// TwinCAT 3 PLC project SystemControl
// Title: Tk_SystemControl
// Company: Komatsu
// Author: TK
// ProjectVersion: 0.0.5.0
// Description: システムの管理用ライブラリ パーシステントデータ管理、PC電源管理
// ProgramVersion: 3.1.4026.26
// libraries:
//   Tc2_IoFunctions, * (Beckhoff Automation GmbH)
//   Tc2_Standard, * (Beckhoff Automation GmbH)
//   Tc2_SUPS, * (Beckhoff Automation GmbH)
//   Tc2_System, * (Beckhoff Automation GmbH)
//   Tc2_Utilities, * (Beckhoff Automation GmbH)
//   Tc3_EventLogger, * (Beckhoff Automation GmbH)
// project tree:
//   PcPower/1s_UPS/ FB_1s_UPS_BAPI.TcPOU, FB_1s_UPS_Base.TcPOU, FB_1s_UPS_CX81xx.TcPOU, I_1s_UPS.TcIO
//   PcPower/ FB_PcShutdownController.TcPOU
//   PcPower/UPS/ FB_UPS_Base.TcPOU, FB_UPS_CU81x0_0xx0.TcPOU, I_UPS.TcIO
//   PcPower/[obsolete]/1sUPS/ FB_1sUPS_BAPI.TcPOU, FB_1sUPS_CX81xx.TcPOU, i1sUPS.TcIO
//   PcPower/[obsolete]/ FB_PcPowerManagement.TcPOU
//   PersistentData/ FB_PersistentDataManager.TcPOU (not stored)
//   PersistentData/[obsolete]/ FB_PersistentDataManagement.TcPOU (not stored)
//   Version/ Global_Version.TcGVL
// (motion and I/O tree: see PLC project wago7871664000080)
// real-time tasks:
//   TASK PlcTask: cycle T#10ms, priority 20, ADS port 350

// ---- Version/Global_Version.TcGVL
{attribute 'TcGenerated'}
{attribute 'no-analysis'}
{attribute 'linkalways'}
// This function has been automatically generated from the project information.
VAR_GLOBAL CONSTANT
	{attribute 'const_non_replaced'}
	stLibVersion_Tk_SystemControl : ST_LibVersion := (iMajor := 0, iMinor := 0, iBuild := 5, iRevision := 0, nFlags := 0, sVersion := '0.0.5.0');
END_VAR

// ---- PcPower/1s_UPS/I_1s_UPS.TcIO
INTERFACE I_1s_UPS

METHOD AcknowledgePowerFailDetect
VAR_INPUT
END_VAR
END_METHOD

PROPERTY bPowerFailDetect : BOOL
GET
END_GET
END_PROPERTY

PROPERTY bReady : BOOL
GET
END_GET
END_PROPERTY

PROPERTY e1sUpsState : E_S_UPS_State
GET
END_GET
END_PROPERTY

METHOD Execute
VAR_INPUT
END_VAR
END_METHOD

//FB_Init は常に暗黙的に使用可能で、主に初期化に使用されます。
//戻り値は評価されません。特定の結果を得るために、メソッドを明示的に宣言し、
//そのメソッドに標準の初期化コードをもったコードを追加することができます。戻り値を評価できます。
METHOD FB_Init: BOOL
VAR_INPUT
    bInitRetains: BOOL; // TRUE: 保持変数は初期化されます (ウォーム リセット、あるいはコールド リセット)
    bInCopyCode: BOOL;  // TRUE: 後でコードをコピーする (オンライン変更) ために、インスタンスをコピーします。

	PcAmsNetId					:AMSNETID;		//PC AMS Net ID
END_VAR
END_METHOD

END_INTERFACE

// ---- PcPower/UPS/I_UPS.TcIO
INTERFACE I_UPS

METHOD AcknowledgePowerFailDetect
VAR_INPUT
END_VAR
END_METHOD

PROPERTY bPowerFailDetect : BOOL
GET
END_GET
END_PROPERTY

PROPERTY bReady : BOOL
GET
END_GET
END_PROPERTY

PROPERTY bReplaceBattery : BOOL
GET
END_GET
END_PROPERTY

METHOD Execute
VAR_INPUT
END_VAR
END_METHOD

//FB_Init は常に暗黙的に使用可能で、主に初期化に使用されます。
//戻り値は評価されません。特定の結果を得るために、メソッドを明示的に宣言し、
//そのメソッドに標準の初期化コードをもったコードを追加することができます。戻り値を評価できます。
METHOD FB_Init: BOOL
VAR_INPUT
    bInitRetains: BOOL; // TRUE: 保持変数は初期化されます (ウォーム リセット、あるいはコールド リセット)
    bInCopyCode: BOOL;  // TRUE: 後でコードをコピーする (オンライン変更) ために、インスタンスをコピーします。

	PcAmsNetId					:AMSNETID;		//PC AMS Net ID
END_VAR
END_METHOD

PROPERTY nBatteryPercent : DWORD
GET
END_GET
END_PROPERTY

END_INTERFACE

// ---- PcPower/[obsolete]/1sUPS/i1sUPS.TcIO
INTERFACE i1sUPS

PROPERTY bPowerFailDetect : bool
GET
END_GET
END_PROPERTY

PROPERTY eUpsState : E_S_UPS_State
GET
END_GET
END_PROPERTY

METHOD UPSCall
VAR_INPUT
	(*PC AMS Net ID*)
	PcAmsNetId	: AMSNETID;
END_VAR
END_METHOD

END_INTERFACE

// ---- PcPower/1s_UPS/FB_1s_UPS_BAPI.TcPOU
FUNCTION_BLOCK FB_1s_UPS_BAPI EXTENDS FB_1s_UPS_Base
VAR CONSTANT
	nOkCapacityLevel	:BYTE	:=90;
END_VAR
VAR
	fb1sUps				:FB_S_UPS_BAPI;
END_VAR

METHOD Execute
fb1sUps(sNetID				:=F_CreateAmsNetId(_PcAmsNetId),
		iPLCPort			:=TwinCAT_SystemInfoVarList._AppInfo.AdsPort,
		tTimeout			:=DEFAULT_ADS_TIMEOUT,
		eUpsMode			:=E_S_UPS_Mode.eSUPS_WrPersistData_Shutdown,
		ePersistentMode		:=E_PersistentMode.SPDM_2PASS,
		tRecoverTime		:=T#10S,
		bPowerFailDetect	=>,
		eState				=>SUPER^._e1sUpsState,
		nCapacity			=>,
		bBusy				=>,
		bError				=>,
		nErrID				=>
		);
		
IF fb1sUps.bPowerFailDetect THEN
	SUPER^._bPowerFailDetect:=TRUE;
END_IF

SUPER^._bReady:=(fb1sUps.eState=E_S_UPS_State.eSUPS_PowerOK) AND (nOkCapacityLevel<fb1sUps.nCapacity) AND (fb1sUps.bError=FALSE);
END_METHOD

END_FUNCTION_BLOCK

// ---- PcPower/1s_UPS/FB_1s_UPS_Base.TcPOU
FUNCTION_BLOCK FB_1s_UPS_Base IMPLEMENTS I_1s_UPS
VAR
	_PcAmsNetId				:AMSNETID;			//PC AMS Net ID	
	
	_bReady					:BOOL;				//電源供給あり
	_e1sUpsState			:E_S_UPS_State;		//1s UPSのステータス
	
	{attribute 'TcPersistent'}
	_bPowerFailDetect		:BOOL;				//停電検知記憶
END_VAR

METHOD AcknowledgePowerFailDetect
_bPowerFailDetect:=FALSE;
END_METHOD

PROPERTY bPowerFailDetect : BOOL
GET
bPowerFailDetect:=_bPowerFailDetect;
END_GET
END_PROPERTY

PROPERTY bReady : BOOL
GET
bReady:=_bReady;
END_GET
END_PROPERTY

PROPERTY e1sUpsState : E_S_UPS_State
GET
e1sUpsState:=_e1sUpsState;
END_GET
END_PROPERTY

METHOD Execute
END_METHOD

//FB_Init は常に暗黙的に使用可能で、主に初期化に使用されます。
//戻り値は評価されません。特定の結果を得るために、メソッドを明示的に宣言し、
//そのメソッドに標準の初期化コードをもったコードを追加することができます。戻り値を評価できます。
METHOD FB_Init: BOOL
VAR_INPUT
    bInitRetains: BOOL; // TRUE: 保持変数は初期化されます (ウォーム リセット、あるいはコールド リセット)
    bInCopyCode: BOOL;  // TRUE: 後でコードをコピーする (オンライン変更) ために、インスタンスをコピーします。

	PcAmsNetId					:AMSNETID;		//PC AMS Net ID
END_VAR
_PcAmsNetId:=PcAmsNetId;
END_METHOD

END_FUNCTION_BLOCK

// ---- PcPower/1s_UPS/FB_1s_UPS_CX81xx.TcPOU
FUNCTION_BLOCK FB_1s_UPS_CX81xx EXTENDS FB_1s_UPS_Base
VAR
	fb1sUps		:FB_S_UPS_CX81xx;
END_VAR

METHOD Execute
fb1sUps(sNetID				:=F_CreateAmsNetId(_PcAmsNetId),
		iPLCPort			:=TwinCAT_SystemInfoVarList._AppInfo.AdsPort,
		tTimeout			:=DEFAULT_ADS_TIMEOUT,
		eUpsMode			:=E_S_UPS_Mode.eSUPS_WrPersistData_Shutdown,
		ePersistentMode		:=E_PersistentMode.SPDM_2PASS,
		tRecoverTime		:=T#10S,
		bPowerFailDetect	=>,
		eState				=>SUPER^._e1sUpsState
		);

IF fb1sUps.bPowerFailDetect THEN
	SUPER^._bPowerFailDetect:=TRUE;
END_IF

SUPER^._bReady:= fb1sUps.eState=E_S_UPS_State.eSUPS_PowerOK;
END_METHOD

END_FUNCTION_BLOCK

// ---- PcPower/FB_PcShutdownController.TcPOU
FUNCTION_BLOCK FB_PcShutdownController
VAR
//---FB_Initで受け取り---
	_pPersistentDataManager		:POINTER TO FB_PersistentDataManager;		//パーシステントデータ書き込み
	_PcAmsNetId					:AMSNETID;									//PC AMS Net ID	

//---内部使用FB---
	fbPlcStop					:PLC_Stop		:=(Stop:=FALSE);			//PLCストップ
	fbNtShutdown				:NT_Shutdown	:=(START:=FALSE);			//PCシャットダウン
	fbNtReboot					:NT_Reboot		:=(START:=FALSE);			//PCリブート

	fbRebootTon					:TON			:=(PT:=T#2S);
	fbShutdownTon				:TON			:=(PT:=T#2S);
	
//---内部変数---
	iStep						:INT			:=0;						//シャットダウン、リブート制御step
	_bError						:BOOL;
	_bReboot					:BOOL;
	_bShutdown					:BOOL;
END_VAR

PROPERTY bError : BOOL
GET
bError:=_bError;
END_GET
END_PROPERTY

METHOD Execute
//---パーシステントデータ保存FBのポインターチェック---
	IF _pPersistentDataManager=0 THEN
		_bError:=TRUE;
		iStep:=0;
		RETURN;
		
	END_IF	



//---タイマーFB呼び出し---
	fbRebootTon(IN:=_bReboot AND NOT _bShutdown AND NOT _bError );
	fbShutdownTon(IN:=_bShutdown AND NOT _bReboot AND NOT _bError );



//---制御step---
	CASE iStep OF
		0:
			IF fbRebootTon.Q OR fbShutdownTon.Q THEN
				iStep:=10;
				
			END_IF
			
		10:				
			_pPersistentDataManager^.RequestWrite();
			iStep:=20;
	
		20:
			IF _pPersistentDataManager^.bWritePersistentDataDone THEN
				iStep:=30;
			ELSIF _pPersistentDataManager^.bWritePersistentDataError THEN
				_bError:=TRUE;
				iStep:=0;
			END_IF
		
		30:
		(*	fbPlcStop(	NETID	:=F_CreateAmsNetId(_PcAmsNetId),
						PORT	:=TwinCAT_SystemInfoVarList._AppInfo.AdsPort,
						Stop	:=_bReboot OR _bShutdown,
						TMOUT	:=DEFAULT_ADS_TIMEOUT,
						BUSY	=>,
						ERR		=>,
						ERRID	=>
						);
		*)
		
			fbNtReboot(	NETID	:=F_CreateAmsNetId(_PcAmsNetId),
						DELAY	:=1,
						START	:=_bReboot,
						TMOUT	:=DEFAULT_ADS_TIMEOUT,
						BUSY	=>,
						ERR		=>,
						ERRID	=>
						);
		
			fbNtShutdown(	NETID	:=F_CreateAmsNetId(_PcAmsNetId),
							DELAY	:=1,
							START	:=_bShutdown,
							TMOUT	:=DEFAULT_ADS_TIMEOUT,
							BUSY	=>,
							ERR		=>,
							ERRID	=>
							);
	
	END_CASE
END_METHOD

//FB_Init は常に暗黙的に使用可能で、主に初期化に使用されます。
//戻り値は評価されません。特定の結果を得るために、メソッドを明示的に宣言し、
//そのメソッドに標準の初期化コードをもったコードを追加することができます。戻り値を評価できます。
METHOD FB_Init: BOOL
VAR_INPUT
    bInitRetains: BOOL; // TRUE: 保持変数は初期化されます (ウォーム リセット、あるいはコールド リセット)
    bInCopyCode: BOOL;  // TRUE: 後でコードをコピーする (オンライン変更) ために、インスタンスをコピーします。

    pPersistentDataManager		:POINTER TO FB_PersistentDataManager;
	PcAmsNetId					:AMSNETID;		//PC AMS Net ID
END_VAR
_pPersistentDataManager := pPersistentDataManager;

_PcAmsNetId:=PcAmsNetId;
END_METHOD

METHOD  RequestReboot: BOOL
VAR_INPUT
	bExecute	:bool;
END_VAR
_bReboot		:=bExecute;
RequestReboot	:=bExecute;
END_METHOD

METHOD RequestShutdown: BOOL
VAR_INPUT
	bExecute	:BOOL;
END_VAR
_bShutdown			:=bExecute;
RequestShutdown		:=bExecute;
END_METHOD

METHOD ResetError
//エラー出力をリセット
_bError:=FALSE;
END_METHOD

END_FUNCTION_BLOCK

// ---- PcPower/UPS/FB_UPS_Base.TcPOU
FUNCTION_BLOCK FB_UPS_Base IMPLEMENTS I_UPS
VAR
	_PcAmsNetId				:AMSNETID;			//PC AMS Net ID	
	
	_bReady					:BOOL;				//電源供給あり
	_bReplaceBattery		:BOOL;				//バッテリー寿命・交換警告
	
	_nBatteryPercent		:DWORD;				//バッテリー残量 (0-100%)
	
	{attribute 'TcPersistent'}
	_bPowerFailDetect		:BOOL;				//停電検知記憶
END_VAR

METHOD AcknowledgePowerFailDetect
_bPowerFailDetect:=FALSE;
END_METHOD

PROPERTY bPowerFailDetect : BOOL
GET
bPowerFailDetect:=_bPowerFailDetect;
END_GET
END_PROPERTY

PROPERTY bReady : BOOL
GET
bReady:=_bReady;
END_GET
END_PROPERTY

PROPERTY bReplaceBattery : BOOL
GET
bReplaceBattery:=_bReplaceBattery;
END_GET
END_PROPERTY

METHOD Execute
END_METHOD

(*FB_Init は常に暗黙的に使用可能で、主に初期化に使用されます。
戻り値は評価されません。特定の結果を得るために、メソッドを明示的に宣言し、
そのメソッドに標準の初期化コードをもったコードを追加することができます。戻り値を評価できます。*)
METHOD FB_Init : BOOL
VAR_INPUT
	(* TRUE: 保持変数は初期化されます (ウォーム リセット、あるいはコールド リセット)*)
	bInitRetains	: BOOL;
	(* TRUE: 後でコードをコピーする (オンライン変更) ために、インスタンスをコピーします。*)
	bInCopyCode	: BOOL;
	(*PC AMS Net ID*)
	PcAmsNetId	: AMSNETID;
END_VAR
_PcAmsNetId:=PcAmsNetId;
END_METHOD

PROPERTY nBatteryPercent : DWORD
GET
nBatteryPercent:=_nBatteryPercent;
END_GET
END_PROPERTY

END_FUNCTION_BLOCK

// ---- PcPower/UPS/FB_UPS_CU81x0_0xx0.TcPOU
FUNCTION_BLOCK FB_UPS_CU81x0_0xx0 EXTENDS FB_UPS_Base
VAR_INPUT
END_VAR
VAR_OUTPUT
END_VAR
VAR
	fbUps			:FB_GetUPSStatus;
	_stUpsStatus	:ST_UPSStatus;
END_VAR

METHOD Execute
fbUps(	sNetId		:=SUPER^._PcAmsNetId,
		nPort		:=0,
		bEnable		:=TRUE,
		bValid		=>,
		bError		=>,
		nErrId		=>,
		stStatus	=>_stUpsStatus
		);

SUPER^._bReady:= fbUps.stStatus.ePowerStatus=E_UpsPowerStatus.PowerOnLine;

SUPER^._bPowerFailDetect:= fbUps.stStatus.ePowerStatus=E_UpsPowerStatus.PowerOnBattery;

SUPER^._bReplaceBattery:=fbUps.stStatus.eBatteryStatus=E_BatteryStatus.BatteryReplace;

SUPER^._nBatteryPercent:=fbUps.stStatus.BatteryLifePercent;
END_METHOD

PROPERTY stUpsStatus : ST_UPSStatus
GET
stUpsStatus:=_stUpsStatus;
END_GET
END_PROPERTY

END_FUNCTION_BLOCK

// ---- PcPower/[obsolete]/1sUPS/FB_1sUPS_BAPI.TcPOU
FUNCTION_BLOCK FB_1sUPS_BAPI IMPLEMENTS i1sUPS
VAR
	fb1sUps		:FB_S_UPS_BAPI;
END_VAR

PROPERTY bPowerFailDetect : BOOL
GET
bPowerFailDetect:=fb1sUps.bPowerFailDetect;
END_GET
END_PROPERTY

PROPERTY eUpsState : E_S_UPS_State
GET
eUpsState := fb1sUps.eState;
END_GET
END_PROPERTY

METHOD UPSCall
VAR_INPUT
	(*PC AMS Net ID*)
	PcAmsNetId	: AMSNETID;
END_VAR
fb1sUps(sNetID				:=F_CreateAmsNetId(PcAmsNetId),
		iPLCPort			:=_AppInfo.AdsPort,
		tTimeout			:=DEFAULT_ADS_TIMEOUT,
		eUpsMode			:=E_S_UPS_Mode.eSUPS_WrPersistData_Shutdown,
		ePersistentMode		:=E_PersistentMode.SPDM_2PASS,
		tRecoverTime		:=T#10S,
		bPowerFailDetect	=>,
		eState				=>,
		nCapacity			=>,
		bBusy				=>,
		bError				=>,
		nErrID				=>
		);
END_METHOD

END_FUNCTION_BLOCK

// ---- PcPower/[obsolete]/1sUPS/FB_1sUPS_CX81xx.TcPOU
FUNCTION_BLOCK FB_1sUPS_CX81xx IMPLEMENTS i1sUPS
VAR
	fb1sUps		:FB_S_UPS_CX81xx;
END_VAR

PROPERTY bPowerFailDetect : BOOL
GET
bPowerFailDetect:=fb1sUps.bPowerFailDetect;
END_GET
END_PROPERTY

PROPERTY eUpsState : E_S_UPS_State
GET
eUpsState := fb1sUps.eState;
END_GET
END_PROPERTY

METHOD UPSCall
VAR_INPUT
	(*PC AMS Net ID*)
	PcAmsNetId	: AMSNETID;
END_VAR
fb1sUps(sNetID				:=F_CreateAmsNetId(PcAmsNetId),
		iPLCPort			:=_AppInfo.AdsPort,
		tTimeout			:=DEFAULT_ADS_TIMEOUT,
		eUpsMode			:=E_S_UPS_Mode.eSUPS_WrPersistData_Shutdown,
		ePersistentMode		:=E_PersistentMode.SPDM_2PASS,
		tRecoverTime		:=T#10S,
		bPowerFailDetect	=>,
		eState				=>
		);
END_METHOD

END_FUNCTION_BLOCK

// ---- PcPower/[obsolete]/FB_PcPowerManagement.TcPOU
FUNCTION_BLOCK FB_PcPowerManagement
VAR
	fbWritePersistentData		:FB_WritePersistentData;	//パーシステントデータ書き込み
	
	fbPlcStop					:PLC_Stop;					//PLCストップ
	
	fbNtShutdown				:NT_Shutdown;				//PCシャットダウン
	fbNtReboot					:NT_Reboot;					//PCリブート
	
	fb1sUPS						:i1sUPS;					//1sUPS管理FB
	
	PcAmsNetId					:AMSNETID;					//PC AMS Net ID
	
	fbRebootTon					:TON;
	fbShutdownTon				:TON;
	
	iRebootStep					:INT;
	iShutdownStep				:INT;
END_VAR
VAR PERSISTENT
	bPowerFailDetected			:BOOL;						//停電検知記憶
END_VAR

//FB_Init は常に暗黙的に使用可能で、主に初期化に使用されます。
//戻り値は評価されません。特定の結果を得るために、メソッドを明示的に宣言し、
//そのメソッドに標準の初期化コードをもったコードを追加することができます。戻り値を評価できます。
METHOD FB_Init: BOOL
VAR_INPUT
    bInitRetains: BOOL; // TRUE: 保持変数は初期化されます (ウォーム リセット、あるいはコールド リセット)
    bInCopyCode: BOOL;  // TRUE: 後でコードをコピーする (オンライン変更) ために、インスタンスをコピーします。

	PcAmsNetId			:AMSNETID;		//PC AMS Net ID
	fb1sUPS				:i1sUPS;
END_VAR
THIS^.PcAmsNetId		:=PcAmsNetId;
THIS^.fb1sUPS			:=fb1sUPS;
END_METHOD

METHOD Reboot
VAR_INPUT
	bReboot	:bool;
END_VAR
CASE iRebootStep OF
	0:
		fbRebootTon(IN:=bReboot,PT:=T#2S,Q=>,ET=>);
			
		IF fbRebootTon.Q=TRUE THEN
			fbWritePersistentData.START:=TRUE;
			iRebootStep:=1;			
		END_IF

	1:
		fbWritePersistentData(	NETID	:=F_CreateAmsNetId(PcAmsNetId),
								PORT	:=_AppInfo.AdsPort,
								START	:=,
								TMOUT	:=DEFAULT_ADS_TIMEOUT,
								MODE	:=E_PersistentMode.SPDM_2PASS,
								BUSY	=>,
								ERR		=>,
								ERRID	=>
								);
	
		IF fbWritePersistentData.BUSY=FALSE THEN
			fbWritePersistentData.START:=FALSE;
			iRebootStep:=2;
		END_IF
	
	2:
		fbPlcStop.STOP:=TRUE;
		fbNtReboot.START:=TRUE;
		iRebootStep:=3;
	
	3:
		fbPlcStop(	NETID	:=F_CreateAmsNetId(PcAmsNetId),
					PORT	:=_AppInfo.AdsPort,
					Stop	:=,
					TMOUT	:=DEFAULT_ADS_TIMEOUT,
					BUSY	=>,
					ERR		=>,
					ERRID	=>
					);

		fbNtReboot(	NETID	:=F_CreateAmsNetId(PcAmsNetId),
					DELAY	:=1,
					START	:=,
					TMOUT	:=DEFAULT_ADS_TIMEOUT,
					BUSY	=>,
					ERR		=>,
					ERRID	=>
					);

END_CASE
END_METHOD

METHOD Shutdown
VAR_INPUT
	bShutdown	:BOOL;
END_VAR
CASE iShutdownStep OF
	0:
		fbShutdownTon(IN:=bShutdown,PT:=T#2S,Q=>,ET=>);
	
		IF fbShutdownTon.Q=TRUE THEN
			fbWritePersistentData.START:=TRUE;
			iShutdownStep:=1;			
		END_IF

	1:
		fbWritePersistentData(	NETID	:=F_CreateAmsNetId(PcAmsNetId),
								PORT	:=_AppInfo.AdsPort,
								START	:=,
								TMOUT	:=DEFAULT_ADS_TIMEOUT,
								MODE	:=E_PersistentMode.SPDM_2PASS,
								BUSY	=>,
								ERR		=>,
								ERRID	=>
								);
	
		IF fbWritePersistentData.BUSY=FALSE THEN
			fbWritePersistentData.START:=FALSE;
			iShutdownStep:=2;
		END_IF
	
	2:
		fbPlcStop.STOP:=TRUE;
		fbNtShutdown.START:=TRUE;
		iShutdownStep:=3;
	
	3:
		fbPlcStop(	NETID	:=F_CreateAmsNetId(PcAmsNetId),
					PORT	:=_AppInfo.AdsPort,
					Stop	:=,
					TMOUT	:=DEFAULT_ADS_TIMEOUT,
					BUSY	=>,
					ERR		=>,
					ERRID	=>
					);

		fbNtShutdown(	NETID	:=F_CreateAmsNetId(PcAmsNetId),
						DELAY	:=1,
						START	:=,
						TMOUT	:=DEFAULT_ADS_TIMEOUT,
						BUSY	=>,
						ERR		=>,
						ERRID	=>
						);
	
END_CASE
END_METHOD

METHOD UPSControl
VAR_INPUT
	bPowerFailDetectReset		:BOOL;
END_VAR
fb1sUPS.UPSCall(PcAmsNetId:=PcAmsNetId);

IF fb1sUPS.bPowerFailDetect=TRUE THEN
	bPowerFailDetected		:=fb1sUPS.bPowerFailDetect;
ELSIF bPowerFailDetectReset=TRUE THEN
	bPowerFailDetected		:=FALSE;
END_IF
END_METHOD

END_FUNCTION_BLOCK
